{attribute 'qualified_only'}
{attribute 'strict'}
{attribute 'to_string'}
TYPE E_DS402OpMode :
(
    NONE:= 0,
    CALIBRATION:=-1,
    MCS2_OL_SM:=-4,
    PROFILE_POSITION:=1,
    HOMING:=6,
    CSP:=8
) SINT;
END_TYPE

(* stored: Version 1.1.0.1
   DUT E_DS402OpMode: Id {6408c62a-847b-4029-9fed-2620404dcad3} *)
